PROGRAM AlarmLogger
VAR
	iCounter:DINT;
	iMax:DINT;
	alarmTrigger: R_TRIG; 
END_VAR

alarmTrigger(CLK := GVL.bCriticalAlarm);

IF alarmTrigger.Q THEN
	//Shift the whole array by 1 so we can enter the new alarm in the first element
	iCounter:=0;
	
	//Max number of alarms
	//Depends on the array size of GVL.aAlarms
	iMax:=15;
	
	FOR iCounter:=iMax TO 0 BY -1 DO //Notice we're counting backwards so the last element goes away, and the first element is now empty
		
		IF iCounter<>iMax THEN
			GVL.aAlarms[iCounter+1]:=GVL.aAlarms[iCounter];
		END_IF	

	END_FOR

	GVL.aAlarms[0].sAlarmText:=GVL.sAlarmText;
	GVL.aAlarms[0].dtTime:=SYSTEMTIME_TO_STRING(GVL.fbLocalSystemTime.systemTime);
	
	GVL.bActiveAlarm:=TRUE; //An alarm is now active and will remain that way until the user acknowledges it

END_IF

END_PROGRAM

(* stored: Version 1.1.0.1, ProductVersion 3.1.4022.16
   POU AlarmLogger: Id {f9349e5e-952a-4c39-92af-9f961481e0a9}, SpecialFunc None *)
